FUNCTION_BLOCK PicAlpha EXTENDS BaseCarrier
VAR_INPUT
END_VAR
VAR_OUTPUT
	o_VacuumGripper: VacuumGripper;
	o_MonostableCylinder: MonostableCylinder;
	o_Distance: INT := 50;
END_VAR
VAR
	m_PresenceSensorPosition1: PresenceSensor;
	m_PresenceSensorPosition2: PresenceSensor;
	m_PresenceSensorPosition3: PresenceSensor;
	m_PresenceSensorPosition4: PresenceSensor;

END_VAR

METHOD METH_CarrierBackward : BOOL
VAR_INPUT
END_VAR
Motor.ACT_TurnCounterclockwise();

IF m_PresenceSensorPosition1.Value THEN
	o_Distance := 0;
ELSIF m_PresenceSensorPosition2.Value THEN
	o_Distance := 10;
ELSIF m_PresenceSensorPosition3.Value THEN
	o_Distance := 50;
ELSIF m_PresenceSensorPosition4.Value THEN
	o_Distance := 100;
END_IF
END_METHOD

METHOD METH_CarrierForward : BOOL
VAR_INPUT
END_VAR
Motor.ACT_TurnClockwise();

IF m_PresenceSensorPosition1.Value THEN
	o_Distance := 0;
ELSIF m_PresenceSensorPosition2.Value THEN
	o_Distance := 10;
ELSIF m_PresenceSensorPosition3.Value THEN
	o_Distance := 50;
ELSIF m_PresenceSensorPosition4.Value THEN
	o_Distance := 100;
END_IF
END_METHOD

METHOD METH_CarrierStop : BOOL
VAR_INPUT
END_VAR
Motor.ACT_Stop();
END_METHOD

PROPERTY PresenceSensorPosition1Value : BOOL
GET
PresenceSensorPosition1Value := m_PresenceSensorPosition1.Value;
END_GET
END_PROPERTY

PROPERTY PresenceSensorPosition2Value : BOOL
GET
PresenceSensorPosition2Value := m_PresenceSensorPosition2.Value;
END_GET
END_PROPERTY

PROPERTY PresenceSensorPosition3Value : BOOL
GET
PresenceSensorPosition3Value := m_PresenceSensorPosition3.Value;
END_GET
END_PROPERTY

PROPERTY PresenceSensorPosition4Value : BOOL
GET
PresenceSensorPosition4Value := m_PresenceSensorPosition4.Value;
END_GET
END_PROPERTY

END_FUNCTION_BLOCK

(* stored: Version 1.1.0.1, ProductVersion 3.1.4024.4
   POU PicAlpha: Id {456e32e4-c200-408e-81a4-d8ce24e5e001}, SpecialFunc None
   Method METH_CarrierBackward: Id {38a2bcc1-1b3b-430a-8238-71dc891884ae}
   Method METH_CarrierForward: Id {b3d35be1-2ca0-49a2-b4fd-41dfbf370514}
   Method METH_CarrierStop: Id {6ae70904-4978-4ec0-94a9-cb1d05b25753}
   Property PresenceSensorPosition1Value: Id {ef8068a8-edb8-4443-8d01-a2dda4e2656c}
   Get Get: Id {f671c29a-5867-4fd9-871a-b150095eb111}
   Property PresenceSensorPosition2Value: Id {56973ba7-97b7-4085-8822-cb17e5ee85df}
   Get Get: Id {d236de1f-28c4-4606-8d89-80543463e961}
   Property PresenceSensorPosition3Value: Id {b29699d7-5acd-45ef-b339-52fe94163248}
   Get Get: Id {7d84c7d6-1e68-4c03-a0ed-3bad4ecbb3c0}
   Property PresenceSensorPosition4Value: Id {86d4402e-6d36-4ce5-8973-3b01add9737f}
   Get Get: Id {304e5126-9b7d-4baf-90c3-1dd066908a02} *)
